TYPE ST_Plant :
STRUCT
    id : DINT;

    name        : STRING(255);
    description : STRING(1023);

    robots : STRING(1023);
END_STRUCT
END_TYPE

(* stored: Version 1.1.0.1, ProductVersion 3.1.4026.18
   DUT ST_Plant: Id {34a6c284-8b94-4e88-8dd8-7ba518424372} *)
